(* PLC project Tc2_Utilities.FB_GetLicenses Demo, tc3-libraries-kb TwinCAT 3.1 *)
(* stored: creationDateTime 2026-05-10T20:00:00, modificationDateTime 2026-05-10T20:00:00 *)

PROGRAM P_Demo_FB_GetLicenses
  VAR
    fbFB_GetLicenses : FB_GetLicenses;  (* Tc2_Utilities.FB_GetLicenses 实例 *)
    arg_bExecute : BOOL;  (* VAR_INPUT bExecute *)
    arg_tTimeout : TIME;  (* VAR_INPUT tTimeout *)
    arg_sNetId : T_AmsNetId;  (* VAR_INPUT sNetId *)
    out_bBusy : BOOL;  (* VAR_OUTPUT bBusy *)
    out_bError : BOOL;  (* VAR_OUTPUT bError *)
    out_nErrorId : UDINT;  (* VAR_OUTPUT nErrorId *)
    out_nValidLicenses : UDINT;  (* VAR_OUTPUT nValidLicenses *)
    out_aValidLicenses : ARRAY[1..nMaxLicenses] OF ST_TcOnlineLicenseInfoData;  (* VAR_OUTPUT aValidLicenses *)
    out_nInvalidLicenses : UDINT;  (* VAR_OUTPUT nInvalidLicenses *)
    out_aInvalidLicenses : ARRAY[1..nMaxLicenses] OF ST_TcOnlineLicenseInfoData;  (* VAR_OUTPUT aInvalidLicenses *)
  END_VAR

            // ============================================================
// Tc2_Utilities.FB_GetLicenses 演示程序（FB 实例）
// ============================================================
// 验证步骤：
//   1. 引用 Tc2_Utilities（及依赖类型所在库 Tc2_System 等）
//   2. 编译 + 登录
//   3. 按 doc.md 给 arg_* 赋值
//   4. 在线监视 out_* / io_* 输出
// ============================================================

fbFB_GetLicenses(
    bExecute := arg_bExecute,
    tTimeout := arg_tTimeout,
    sNetId := arg_sNetId,
    bBusy => out_bBusy,
    bError => out_bError,
    nErrorId => out_nErrorId,
    nValidLicenses => out_nValidLicenses,
    aValidLicenses => out_aValidLicenses,
    nInvalidLicenses => out_nInvalidLicenses,
    aInvalidLicenses => out_aInvalidLicenses
);

          
END_PROGRAM
